% RSLogix 500 project UN1.RSS, saved by version 8.10.00.18 %
PROJECT "UN1"    % processor: MicroLogix 1200 %

PROGRAM FILES
  LAD 2   5 rungs

DATA FILES
  O0 OUTPUT  4 elements
  I1 INPUT  4 elements
  S2 STATUS  66 elements
  B3 BINARY  1 elements
  T4 TIMER  1 elements
  C5 COUNTER  1 elements
  R6 CONTROL  1 elements
  N7 INTEGER  1 elements

LADDER 2
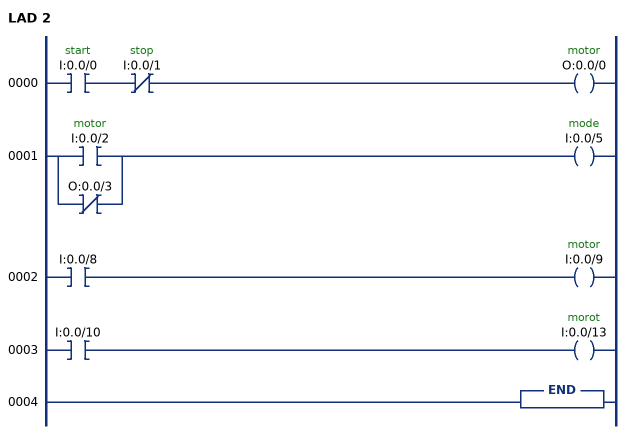
% Rung: 0 %  % edit flag set %
SOR XIC I:0.0/0 XIO I:0.0/1 OTE O:0.0/0 EOR
%   I:0.0/0  "start" %
%   I:0.0/1  "stop" %
%   O:0.0/0  "motor" %
% Rung: 1 %  % edit flag set %
SOR BST XIC I:0.0/2 NXB XIO O:0.0/3 BND OTE I:0.0/5 EOR
%   I:0.0/2  "motor" %
%   I:0.0/5  "mode" %
% Rung: 2 %  % edit flag set %
SOR XIC I:0.0/8 OTE I:0.0/9 EOR
%   I:0.0/9  "motor" %
% Rung: 3 %  % edit flag set %
SOR XIC I:0.0/10 OTE I:0.0/13 EOR
%   I:0.0/13  "morot" %
% Rung: 4 %
SOR END EOR
